	16#4B75: sMsg := '4B75 parameter ST_NciTangentialFollowingDesc: nPathAxis1 and nPathAxis2, resp. are no path axes. So it is not possible to determine the plane.';
	16#4B76: sMsg := '4B76 parameter ST_NciTangentialFollwoingDesc: nPathAxis1 and nPathAxis2 are equal. So it is not possible to determine the plane.';
	16#4B77: sMsg := '4B77 parameter ST_NciGeoCirclePlane: circle is programmed in a wrong manner.';
	16#4B78: sMsg := '4B78 function Internal error in calculation of the tangential following';
	16#4B79: sMsg := '4B79 monitoring Tangential following: With ST_NciTangentialFollowingDesc the monitoring of the deviation angle (E_TfErrorOnCrirical1) is activated and with the actual segment the deviation angle is too big.';
	16#4B7A: sMsg := '4B7A function not implemented';
	16#4B7B: sMsg := '4B7B parameter Tangential Following: The radius of the actual circle segment is too small';
	16#4B7C: sMsg := '4B7C parameter FB_NciFeedTablePreparation: pEntry is NULL';
	16#4B7D: sMsg := '4B7D parameter FB_NciFeedTablePreparation: The specified nEntryType does not match the the structure type';
	16#4B7E: sMsg := '4B7E parameter ST_NciMFuncFast and ST_NciMFuncHsk: The requested m-function is not in between 0..159';
	16#4B7F: sMsg := '4B7F parameter ST_NciDynOvr: The requested value for the dynamic override is not in between 0.01 and 1.0';
	16#4B80: sMsg := '4B80 parameter ST_NciVertexSmoothing: invalid parameter. This error occurs with a negative vertex radius or an unknown vertex smoothing type.';
	16#4B81: sMsg := '4B81 parameter FB_NciFeedTablePrepartion: The requested velocity is not in a valid range';
	16#4B82: sMsg := '4B82 parameter ST_Nci*: invalid parameter';

ELSE
	sMsg := UDINT_TO_STRING(iErrID);
	sMsg := concat(sMsg, ' Unknown Error code');
END_CASE
F_AxErrMsg := sMsg;

END_FUNCTION

(* stored: Version 1.1.0.1, ProductVersion 3.1.4022.16
   POU F_AxErrMsg: Id {06508107-56b8-4212-aec4-06150cd92788}, SpecialFunc None *)
